FUNCTION_BLOCK FB_TestFb1
VAR_INPUT
END_VAR
VAR_OUTPUT
END_VAR
VAR
END_VAR

END_FUNCTION_BLOCK

(* stored: Version 1.1.0.1, ProductVersion 3.1.4024.12
   POU FB_TestFb1: Id {6549275c-2b52-4de2-b628-949c68a66d43}, SpecialFunc None *)
